// TIA Portal V20 export
DATA_BLOCK "BK23"   // DB270
// stored: MemoryReserve 100
   VAR
      "X10-1 JR Unloading P&P Y-AXIS LIMIT SENSOR(-)" : Bool;
      "X11-1 JR Unloading P&P Y-AXIS LIMIT SENSOR(+)" : Bool;
      "X12-1 JR Unloading P&P Z-AXIS LIMIT SENSOR(-)" : Bool;
      "X13-1 JR Unloading P&P Z-AXIS LIMIT SENSOR(+)" : Bool;
      "X14-1 JR Unloading P&P C-AXIS LIMIT SENSOR(-)" : Bool;
      "X15-1 JR Unloading P&P C-AXIS LIMIT SENSOR(+)" : Bool;
      "X16-1 JR Unloading P&P CLAMP OPEN SENSOR" : Bool;
      "X17-1 JR Unloading P&P CLAMP STACK DETECT SENSOR" : Bool;
      "X10-2 JR Unloading P&P Y-AXIS HOMING SENSOR" : Bool;
      "X11-2 SPARE" : Bool;
      "X12-2 JR Unloading P&P Z-AXIS HOMING SENSOR" : Bool;
      "X13-2 SPARE" : Bool;
      "X14-2 JR Unloading P&P C-AXIS HOMING SENSOR" : Bool;
      "X15-2 SPARE" : Bool;
      "X16-2 JR Unloading P&P CLAMP CLOSE SENSOR" : Bool;
      "X17-2 JR Unloading P&P Z-AXIS SAFETY PIN LOADING SENSOR" : Bool;
   END_VAR
BEGIN
END_DATA_BLOCK
